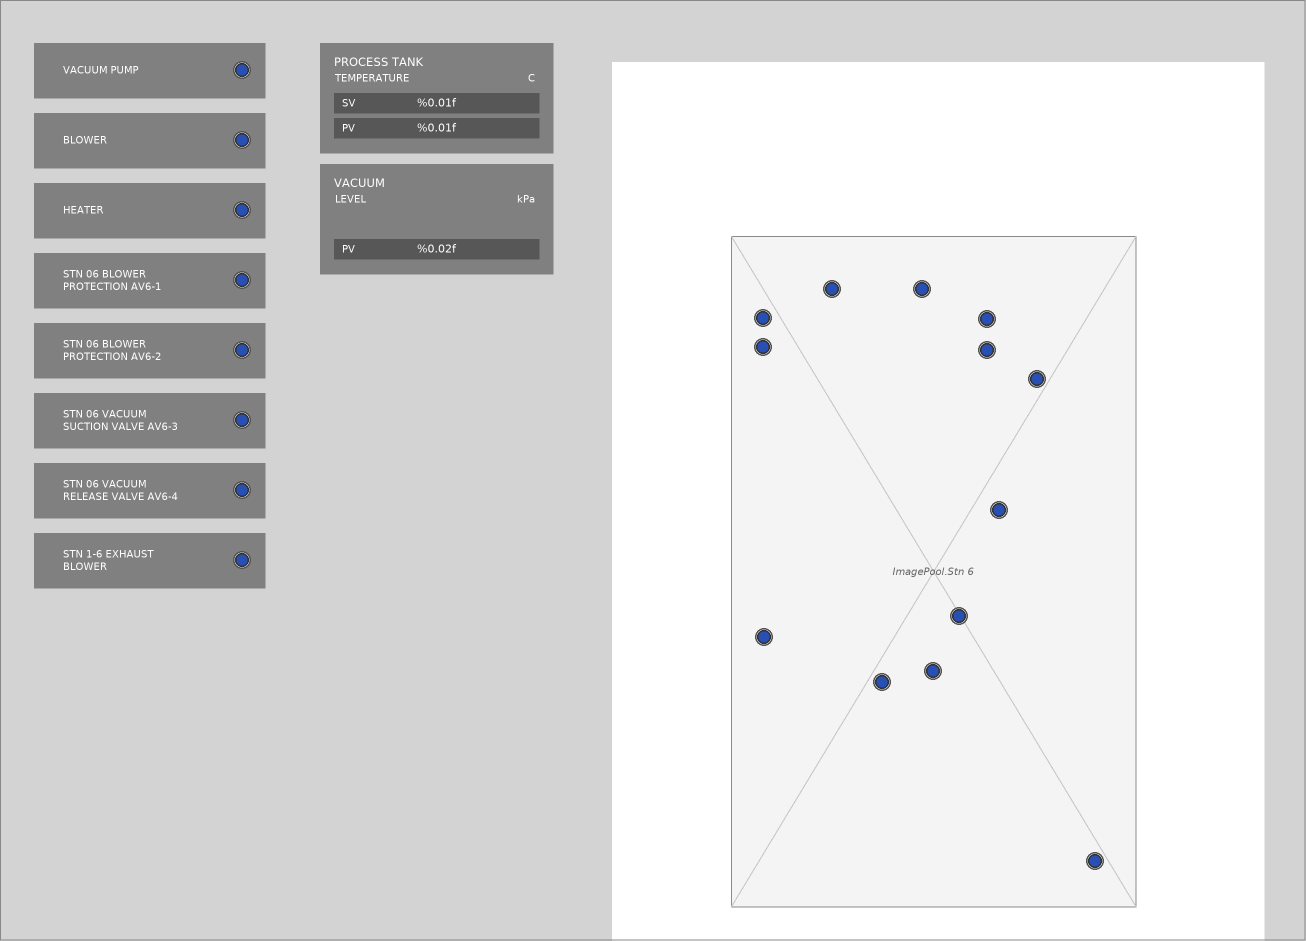
VISUALIZATION Auto_Station06  // 1306x941
    Rectangle (0,0 1306x875)
    RoundedRectangle (34,43 231x55)
    Label (60,62 163x16), "VACUUM PUMP"
    Lamp1 (232,60 20x20), variable: ARdsMAP_HmiVariableStn[6].bProTankVacuumPump_IND, style: Lamp-Lamp1-Blue
    RoundedRectangle (34,113 231x55)
    Label (60,132 151x16), "BLOWER"
    Lamp1 (232,130 20x20), variable: ARdsMAP_HmiVariableStn[6].bProTankBlower_IND, style: Lamp-Lamp1-Blue
    RoundedRectangle (34,183 231x55)
    Label (60,202 151x16), "HEATER"
    Lamp1 (232,200 20x20), variable: ARdsMAP_HmiVariableStn[6].bProTankHeater_IND, style: Lamp-Lamp1-Blue
    RoundedRectangle (34,253 231x55)
    Lamp1 (232,270 20x20), variable: ARdsMAP_HmiVariableStn[6].bValve01_IND, style: Lamp-Lamp1-Blue
    RoundedRectangle (320,43 233x110)
    Label (331,54 150x16), "PROCESS TANK"
    Label (332,67 99x22), "TEMPERATURE"
    Label (509,67 29x22), "C"
    Rectangle (334,93 205x20), "%0.01f", text variable: ARrStnTempSV[6]
    Label (339,92 22x22), "SV"
    Rectangle (334,118 205x20), "%0.01f", text variable: ARrStnTempPV[6]
    Label (339,117 22x22), "PV"
    RoundedRectangle (320,164 233x110)
    Label (331,175 150x16), "VACUUM"
    Label (332,188 99x22), "LEVEL"
    Label (509,188 29x22), "kPa"
    Rectangle (334,239 205x20), "%0.02f", text variable: ARrStnVacuumPV[6]
    Label (339,238 22x22), "PV"
    Label (60,267 151x27), "STN 06 BLOWER PROTECTION AV6-1"
    RoundedRectangle (34,323 231x55)
    Lamp1 (232,340 20x20), variable: ARdsMAP_HmiVariableStn[6].bValve02_IND, style: Lamp-Lamp1-Blue
    Label (60,337 151x27), "STN 06 BLOWER PROTECTION AV6-2"
    RoundedRectangle (34,393 231x55)
    Lamp1 (232,410 20x20), variable: ARdsMAP_HmiVariableStn[6].bValve03_IND, style: Lamp-Lamp1-Blue
    Label (60,407 151x27), "STN 06 VACUUM SUCTION VALVE AV6-3"
    RoundedRectangle (34,463 231x55)
    Lamp1 (232,480 20x20), variable: ARdsMAP_HmiVariableStn[6].bValve04_IND, style: Lamp-Lamp1-Blue
    Label (60,477 151x27), "STN 06 VACUUM RELEASE VALVE AV6-4"
    RoundedRectangle (34,533 231x55)
    Lamp1 (232,550 20x20), variable: ARdsMAP_HmiVariableGeneral.bExhaustBlower_IND, style: Lamp-Lamp1-Blue
    Label (60,547 151x27), "STN 1-6 EXHAUST BLOWER"
    Rectangle (612,62 652x879)
    Image (731,236 405x671), image: ImagePool.Stn 6
    Lamp1 (1085,851 20x20), variable: ARdsMAP_HmiVariableStn[6].bProTankVacuumPump_IND, style: Lamp-Lamp1-Blue
    Lamp1 (923,661 20x20), variable: ARdsMAP_HmiVariableStn[6].bProTankBlower_IND, style: Lamp-Lamp1-Blue
    Lamp1 (872,672 20x20), variable: ARdsMAP_HmiVariableStn[6].bProTankHeater_IND, style: Lamp-Lamp1-Blue
    Lamp1 (949,606 20x20), variable: ARdsMAP_HmiVariableStn[6].bValve02_IND, style: Lamp-Lamp1-Blue
    Lamp1 (1027,369 20x20), variable: ARdsMAP_HmiVariableStn[6].bValve04_IND, style: Lamp-Lamp1-Blue
    Lamp1 (989,500 20x20), variable: ARdsMAP_HmiVariableStn[6].bValve03_IND, style: Lamp-Lamp1-Blue
    Lamp1 (754,627 20x20), variable: ARdsMAP_HmiVariableStn[6].bValve01_IND, style: Lamp-Lamp1-Blue
    Lamp1 (753,337 20x20), variable: ARbDI[eX12100_Stn06SlidingDoorRs01_Clamp], style: Lamp-Lamp1-Blue
    Lamp1 (977,340 20x20), variable: ARbDI[eX12102_Stn06SlidingDoorRs02_Clamp], style: Lamp-Lamp1-Blue
    Lamp1 (753,308 20x20), variable: ARbDI[eX12101_Stn06SlidingDoorRs01_Unclamp], style: Lamp-Lamp1-Blue
    Lamp1 (977,309 20x20), variable: ARbDI[eX12103_Stn06SlidingDoorRs02_Unclamp], style: Lamp-Lamp1-Blue
    Lamp1 (912,279 20x20), variable: ARbDI[eX12008_Stn06SlidingDoorRs_Close], style: Lamp-Lamp1-Blue
    Lamp1 (822,279 20x20), variable: ARbDI[eX12007_Stn06SlidingDoorRs_Open], style: Lamp-Lamp1-Blue
END_VISUALIZATION

(* stored: Version 1.1.0.1, ProductVersion 3.1.4024.12
   Visu Auto_Station06: Id {3d092f89-7153-445b-8707-2d26af1f9764} *)
